PROGRAM uloha1
VAR
	stop: bool;
	Motor: bool;
	start: bool;
	stav: INT;
	casovac: TON;
	casovac2: Ton;
	reset: BOOL;
END_VAR

IF reset = TRUE THEN
	stop := FALSE; 
	start := FALSE ;
	stav := 0;
END_IF

CASE stav OF

    0:  
        Motor := FALSE;

        casovac(IN := FALSE, PT := T#5S);
        casovac2(IN := FALSE, PT := T#5S);

        IF start THEN
            stav := 10;
        END_IF;

    10: 
        Motor := TRUE;

        casovac(IN := TRUE, PT := T#5S);     
        casovac2(IN := FALSE, PT := T#5S);   

        IF casovac.Q THEN
            casovac(IN := FALSE, PT := T#5S); 
            stav := 20;
        END_IF;

        IF stop THEN
            stav := 0;
        END_IF;

    20: 
        Motor := FALSE;

        casovac(IN := FALSE, PT := T#5S);
        casovac2(IN := TRUE, PT := T#5S);    

        IF casovac2.Q THEN
            casovac2(IN := FALSE, PT := T#5S); 
            stav := 10;
        END_IF;

        IF stop THEN
            stav := 0;
        END_IF;

END_CASE;

END_PROGRAM

(* stored: Version 1.1.0.1
   POU uloha1: Id {eaccaacd-b563-4f99-b516-834fdc1fdcdf}, SpecialFunc None *)
